FUNCTION atan2 : LREAL
VAR_INPUT
	y:LREAL;
	x:lreal;	
END_VAR
VAR
END_VAR


IF (x>0 AND y>0) THEN  //第1象限
	atan2:=ATAN(y/x);
ELSIF(x<0 AND y>0) THEN  //第2象限
	atan2:=ATAN(y/x)+pi;

ELSIF(x<0 AND y<0) THEN  //第3象限
	atan2:=ATAN(y/x)-pi;

ELSIF(x>0 AND y<0) THEN  //第4象限
	atan2:=ATAN(y/x);

ELSIF (x=0 AND y>0) THEN  //正Y轴
	atan2:=pi/2;

ELSIF (x=0 AND y<0) THEN  //负Y轴
	atan2:=-pi/2;
	
ELSIF (x>0 AND y=0) THEN  //正X轴
	atan2:=0;

ELSIF (x<0 AND y=0) THEN  //负X轴
	atan2:=pi;	
	
END_IF

END_FUNCTION

(* stored: Version 1.1.0.1, ProductVersion 3.1.4024.12
   POU atan2: Id {87ba860d-899f-4cfa-80d6-9dc1deead6f8}, SpecialFunc None *)
